// TIA Portal V19 export
TYPE "lexchangetray_typeroller_signalTM_Interface"
// Type: lexchangetray_typeroller_signalTM_Simulation
// Type: lexchangetray_typeroller_signalTM_Monitor
// Type: lexchangetray_typeroller_signalTM_Cmd
// stored: Access Published
   STRUCT
      cmd : "lexchangetray_typeroller_signalTM_Cmd";
      monitor { S7_SetPoint := 'True'} : "lexchangetray_typeroller_signalTM_Monitor";
      sim { S7_SetPoint := 'True'} : "lexchangetray_typeroller_signalTM_Simulation";
   END_STRUCT;
END_TYPE
